Fanuc KAREL source: ko00061.KL

PROGRAM KO00061
%STACKSIZE=65535
%PRIORITY=65535
%NOLOCKGROUP
VAR
P1 : XYZWPR
P2 : JOINTPOS9
F : BOOLEAN
OUT : POSITION
BEGIN
F=TRUE
-- UNSAFE_SOURCE_IR line 11: CALL_RESULT MIRROR(convert_xyzwpr_to_xyzwprext(P1), convert_jointpos9_to_position(P2), F)
END KO00061
